// TwinCAT 3 PLC project Untitled1
// ProgramVersion: 3.1.4024.0
// libraries:
//   Tc2_Standard, * (Beckhoff Automation GmbH)
//   Tc2_System, * (Beckhoff Automation GmbH)
//   Tc3_Module, * (Beckhoff Automation GmbH)
// project tree:
//   / PlcTask.TcTTO
//   POUs/ FB_LoadBinaryFile.TcPOU, MAIN.TcPOU, VecMulMatFlat.TcPOU, SampleUdpEchoServer.TcPOU
// real-time tasks:
//   TASK PlcTask: cycle T#1ms, priority 20, ADS port 350
// motion (NC):
//   TASK NC-Task 1 SAF: cycle T#2ms, priority 4, ADS port 501
//   TASK NC-Task 1 SVB: cycle T#10ms, priority 8, ADS port 511
// I/O:
//   DEVICE Device 2 (EtherCAT), AmsNetId 169.254.224.240.3.1
//     Term 1 (EK1100) [EK1100 EtherCAT Coupler (2A E-Bus)]
//       Term 2 (EL4078) [EL4078 8Ch. Ana. Output, +/-10V, +/-20mA, 16 Bit]
//       Term 3 (EL4078) [EL4078 8Ch. Ana. Output, +/-10V, +/-20mA, 16 Bit]
//       Term 4 (EL4078) [EL4078 8Ch. Ana. Output, +/-10V, +/-20mA, 16 Bit]
//       Term 5 (EL9011) [EL9011 End Terminal]
//   DEVICE Device 3 (RT-Ethernet Adapter)
// variable links:
//   Untitled1/Untitled1 Instance <-> Device 2 (EtherCAT)/Term 1 (EK1100)/Term 2 (EL4078)
//     PlcTask Outputs/MAIN.udp1.value0 <-> AO Standard (Real32) Channel 1/Value (Real32)
//     PlcTask Outputs/MAIN.udp1.value1 <-> AO Standard (Real32) Channel 2/Value (Real32)

CONFIGURATION Untitled1
    RESOURCE PLC ON TwinCAT3
        TASK PlcTask(INTERVAL := T#1ms, PRIORITY := 20);
        PROGRAM MAIN WITH PlcTask : MAIN;
    END_RESOURCE
END_CONFIGURATION

// ---- POUs/MAIN.TcPOU
PROGRAM MAIN
VAR
	udp1:  SampleUdpEchoServer;
END_VAR


udp1();

END_PROGRAM

// ---- POUs/SampleUdpEchoServer.TcPOU
{attribute 'c++_compatible'}
FUNCTION_BLOCK SampleUdpEchoServer IMPLEMENTS ITcIoUdpProtocolRecv
VAR_INPUT
END_VAR
VAR_OUTPUT
END_VAR
VAR
	{attribute 'TcInitSymbol'}
    oid:              OTCID;
	ipUdp:            ITcIoUdpProtocol;
	nUdpPort:         UINT := 10000;
	nReceivedPackets: UINT;
	hrInit:           HRESULT;
	hrSend:           HRESULT;
	
	
	step:          UINT := 2;
	nModes:           UINT := 185;
	nActs:            UINT := 185;
	
	m2cMatrix:        ARRAY[0..185*185-1] OF REAL;
	m2cFilename:      STRING := 'C:\TwinCAT\3.1\Boot\eye185.bin';
    fbLoad:           FB_LoadBinaryFile;

	counter: UINT := 0;

	value0 AT %Q*:    REAL;
	value1 AT %Q*:    REAL;


	i: INT;
	value: INT;
END_VAR


FOR i := 0 TO 184 DO
	m2cMatrix[i*185+i] := 1.0;
END_FOR;

CASE step OF

0: 
    fbLoad(
      sFileName := m2cFilename,
      pDest := ADR(m2cMatrix),
      cbSize := SIZEOF(m2cMatrix),
      bExecute := TRUE
	);
	step := 1;
	
1:
	IF fbLoad.bDone THEN
		step  := 2;
	END_IF

2: // start listening for UDP packets

	IF ipUdp <> 0 THEN
		ipUdp.CheckReceived();
	END_IF

END_CASE

METHOD FB_exit : BOOL
VAR_INPUT
	bInCopyCode : BOOL; // if TRUE, the exit method is called for exiting an instance that is copied afterwards (online change).
END_VAR
IF (NOT bInCopyCode AND ipUdp <> 0) THEN //Shutdown
     ipUdp.UnregisterReceiver(nUdpPort);
     FW_SafeRelease(ADR(ipUdp));
     FB_exit := TRUE;
ELSE
     FB_exit := FALSE;
END_IF
END_METHOD

METHOD FB_init : BOOL
VAR_INPUT
	bInitRetains : BOOL; // if TRUE, the retain variables are initialized (warm start / cold start)
	bInCopyCode : BOOL;  // if TRUE, the instance afterwards gets moved into the copy code (online change)
END_VAR
IF NOT bInCopyCode THEN // no online change
    IF ipUdp = 0 AND oid <> 0 THEN
     hrInit := FW_ObjMgr_GetObjectInstance(oid:=oid, iid:=TC_GLOBAL_IID_LIST.IID_ITcIoUdpProtocol, pipUnk:=ADR(ipUdp) );
        IF SUCCEEDED(hrInit) THEN 
            IF SUCCEEDED(ipUdp.RegisterReceiver(nUdpPort, THIS^)) THEN //open port
                FB_init := TRUE;
            ELSE 
                FB_init := FALSE; 
                FW_SafeRelease(ADR(ipUdp));
            END_IF
        END_IF
    ELSIF oid = 0 THEN 
        FB_init := FALSE; 
        hrInit := ERR_INVALID_PARAM;                 
    END_IF
END_IF
END_METHOD

METHOD FB_reinit : BOOL
VAR_INPUT
END_VAR
IF (ipUdp <> 0) THEN 
   ipUdp.RegisterReceiver(nUdpPort, THIS^);
   FB_reinit := TRUE;
END_IF
END_METHOD

{attribute 'TcTypeSystem'}
{attribute 'no-analysis'}
{attribute 'c++_compatible'}
{attribute 'minimal_input_size' := '4'}
{attribute 'pack_mode' := '4'}
{warning 'add method implementation '}
METHOD ReceiveData : HRESULT
VAR_INPUT
	ipAddr	: UDINT;
	udpDestPort	: UINT;
	udpSrcPort	: UINT;
	nData	: UDINT;
	pData	: PVOID;
	pVlan	: POINTER TO ETYPE_VLAN_HEADER := 0;
END_VAR

VAR
	dati:  STRING :=  'ciaociao';
	pDati : PVOID :=  0;

	pModes :    POINTER TO ARRAY[0..185-1] OF REAL;	
    Commands :  ARRAY[0..185-1] OF REAL;

END_VAR
nReceivedPackets := nReceivedPackets+1;
//lastReceivedIP.ipadrIPStack := ipAddr;

counter := counter + 1;

pDati := ADR(dati);
IF ipUdp <> 0 THEN
	
	pModes := pData;
	
	VecMulMatFlat(
		pData,
		ADR(m2cMatrix[0]),
    	ADR(Commands[0]),
    	185,
		185,
 	);
	
	// TODO debug modal projection and set outputs
	
//	value0 := Commands[0];
//	value1 := Commands[1];
//	value0 := m2cMatrix[185];
//	value1 := m2cMatrix[186];

	value0 := pModes^[0];
	value1 := pModes^[1];
	
	ipUdp.SendData(ipAddr, udpSrcPort, udpDestPort, 8, pDati, TRUE, 0); // send data back
END_IF
END_METHOD

{attribute 'TcTypeSystem'}
{attribute 'no-analysis'}
{attribute 'c++_compatible'}
{attribute 'minimal_input_size' := '4'}
{attribute 'pack_mode' := '4'}
{warning 'add method implementation '}
METHOD TcAddRef : UDINT
END_METHOD

{attribute 'TcTypeSystem'}
{attribute 'no-analysis'}
{attribute 'c++_compatible'}
{attribute 'minimal_input_size' := '4'}
{attribute 'pack_mode' := '4'}
{warning 'add method implementation '}
METHOD TcQueryInterface : HRESULT
VAR_INPUT
	iid	: REFERENCE TO IID;
	pipItf	: POINTER TO PVOID;
END_VAR
VAR
   ipUdpRecv : ITcIoUdpProtocolRecv;
   ipUnknown : ITcUnknown;   
END_VAR
IF GuidsEqual(ADR(iid), ADR(TC_GLOBAL_IID_LIST.IID_ITcIoUdpProtocolRecv)) THEN
    ipUdpRecv := THIS^; // cast to interface pointer
    pipItf^ := ITCUNKNOWN_TO_PVOID(ipUdpRecv);
    TcAddRef();
    TcQueryInterface := S_OK;
ELSIF GuidsEqual(ADR(iid), ADR(TC_GLOBAL_IID_LIST.IID_ITcUnknown)) THEN
    ipUnknown := THIS^; // cast to interface pointer
    pipItf^ := ITCUNKNOWN_TO_PVOID(ipUnknown);
    TcAddRef();
    TcQueryInterface := S_OK;
ELSE
    TcQueryInterface := E_HRESULTAdsErr.NOINTERFACE ; //Call super if this fb extends some other
END_IF
END_METHOD

{attribute 'TcTypeSystem'}
{attribute 'no-analysis'}
{attribute 'c++_compatible'}
{attribute 'minimal_input_size' := '4'}
{attribute 'pack_mode' := '4'}
{warning 'add method implementation '}
METHOD TcRelease : UDINT
END_METHOD

END_FUNCTION_BLOCK

// ---- POUs/FB_LoadBinaryFile.TcPOU
FUNCTION_BLOCK FB_LoadBinaryFile
VAR_INPUT
    sFileName : T_MaxString;
    pDest     : PVOID;
    cbSize    : UDINT;
    bExecute  : BOOL;
END_VAR

VAR_OUTPUT
    bDone  : BOOL;
    bBusy  : BOOL;
    bError : BOOL;
    nErrId : UDINT;
END_VAR

VAR
    fbOpen  : FB_FileOpen;
    fbRead  : FB_FileRead;
    fbClose : FB_FileClose;

    hFile : UINT;
    step  : INT;
END_VAR




CASE step OF

0: // idle
    IF bExecute THEN
        bBusy := TRUE;
        bDone := FALSE;
        bError := FALSE;
        step := 1;
    END_IF


1: // open file
    fbOpen(
        sNetId := '',
        sPathName := sFileName,
        nMode := FOPEN_MODEREAD OR FOPEN_MODEBINARY,
        bExecute := TRUE
    );

    IF NOT fbOpen.bBusy THEN
        IF fbOpen.bError THEN
            bError := TRUE;
            nErrId := fbOpen.nErrId;
            step := 100;
        ELSE
            hFile := fbOpen.hFile;
            step := 2;
        END_IF
    END_IF


2: // read file
    fbRead(
        sNetId := '',
        hFile := hFile,
        pReadBuff := pDest,
        cbReadLen := cbSize,
        bExecute := TRUE
    );

    IF NOT fbRead.bBusy THEN
        IF fbRead.bError THEN
            bError := TRUE;
            nErrId := fbRead.nErrId;
            step := 100;
        ELSE
            step := 3;
        END_IF
    END_IF


3: // close file
    fbClose(
        sNetId := '',
        hFile := hFile,
        bExecute := TRUE
    );

    IF NOT fbClose.bBusy THEN
        step := 10;
    END_IF


10: // finished
    bBusy := FALSE;
    bDone := TRUE;

    IF NOT bExecute THEN
        step := 0;
    END_IF


100: // error
    bBusy := FALSE;

END_CASE

END_FUNCTION_BLOCK

// ---- POUs/VecMulMatFlat.TcPOU
FUNCTION VecMulMatFlat : BOOL
VAR_INPUT
    pVec    : POINTER TO REAL; // input vector (size N)
    pMat    : POINTER TO REAL; // matrix as flat vector (N*M)
    pRes    : POINTER TO REAL; // result vector (size M)
    nVec    : UDINT;           // vector size
    nCols   : UDINT;           // matrix columns
END_VAR

VAR
    i       : UDINT;
    j       : UDINT;
    sum     : REAL;
    pV      : POINTER TO REAL;
    pM      : POINTER TO REAL;
END_VAR



pM := pMat;

FOR j := 0 TO nCols - 1 DO

    sum := 0.0;
    pV := pVec;

    FOR i := 0 TO nVec - 1 DO

        sum := sum + pV^ * pM^;
        pV := pV + 1;
        pM := pM + 1;
    END_FOR

	pRes[j] := sum;

END_FOR

VecMulMatFlat := TRUE;

END_FUNCTION
